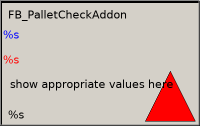
VISUALIZATION V_PalletCheckAddon  // 200x126
VAR_IN_OUT
	{attribute 'VAR_IN_OUT_AS_POINTER'}
	fbFunction		: FB_PalletCheckAddon;
END_VAR
    Rectangle (0,1 200x125)
    Rectangle (5,105 143x20), "%s", text variable: fbFunction.ConfigFunction.FunctionName
    Label (5,5 158x20), "FB_PalletCheckAddon"
    Rectangle (0,25 99x20), "%s", text variable: fbFunction.eState
    Polygon (145,121) (170,71) (195,121) (180,121) (160,121), invisible if: fbFunction.FunctionData.ErrorData.ErrorState = E_ErrorState.OPERATIONAL
    Rectangle (0,50 161x20), "%s", text variable: fbFunction.FunctionData.ErrorData.Error.ErrorCode.Conv, invisible if: fbFunction.FunctionData.ErrorData.Error.ErrorCode.Conv = 0
    Label (7,77 158x15), "show appropriate values here"
END_VISUALIZATION

(* stored: Version 1.1.0.1, ProductVersion 3.1.4024.4
   Visu V_PalletCheckAddon: Id {3572b172-20e8-454f-971a-ade89dbd2f06} *)
